(* PLC project 1000-tech-water, Неизвестно 1000-tech-water 1 *)
(* stored: creationDateTime 2022-06-13T20:45:02, productRelease 0, contentDescription 2022-06-20 Локальные испытания: выполнены Комплексные испытания: выполнены, modificationDateTime 2022-06-20T21:02:03, version 0, language ru-RU *)

PROGRAM Main
  VAR_EXTERNAL
    LT_Low : BOOL;
  END_VAR
  VAR
    LT_Low_f : BOOL;  (* Отфильтрованное значение *)
  END_VAR
  VAR_EXTERNAL
    LT_Middle : BOOL;
  END_VAR
  VAR
    LT_Middle_f : BOOL;  (* Отфильтрованное значение *)
  END_VAR
  VAR_EXTERNAL
    LT_Hight : BOOL;
  END_VAR
  VAR
    LT_Hight_f : BOOL;  (* Отфильтрованное значение *)
  END_VAR
  VAR_EXTERNAL
    HS_Auto : BOOL;
  END_VAR
  VAR
    HS_Auto_f : BOOL;  (* Отфильтрованное значение *)
  END_VAR
  VAR_EXTERNAL
    P_Speed_50 : BOOL;
  END_VAR
  VAR
    P_Speed_50L : BOOL;
  END_VAR
  VAR_EXTERNAL
    P_Speed_100 : BOOL;
  END_VAR
  VAR
    P_Speed_100L : BOOL;
  END_VAR
  VAR_EXTERNAL
    P_Start : BOOL;
  END_VAR
  VAR
    P_StartL : BOOL;
  END_VAR
  VAR_EXTERNAL
    LT_error : BOOL;
  END_VAR
  VAR
    LT_errorL : BOOL;
  END_VAR
  VAR_EXTERNAL
    LT_set : BOOL;
    PLC_state : WORD;
  END_VAR
  VAR
    TON0 : TON;
  END_VAR
  VAR CONSTANT
    TM_5S : TIME := T#5s;  (* Время 5 сек *)
  END_VAR
  VAR
    TON1 : TON;
    TON2 : TON;
    TON3 : TON;
  END_VAR
  VAR  (* added by the conversion: wires and edge detectors of the diagram *)
    _OR68_OUT : BOOL;
    _OR58_OUT : BOOL;
  END_VAR

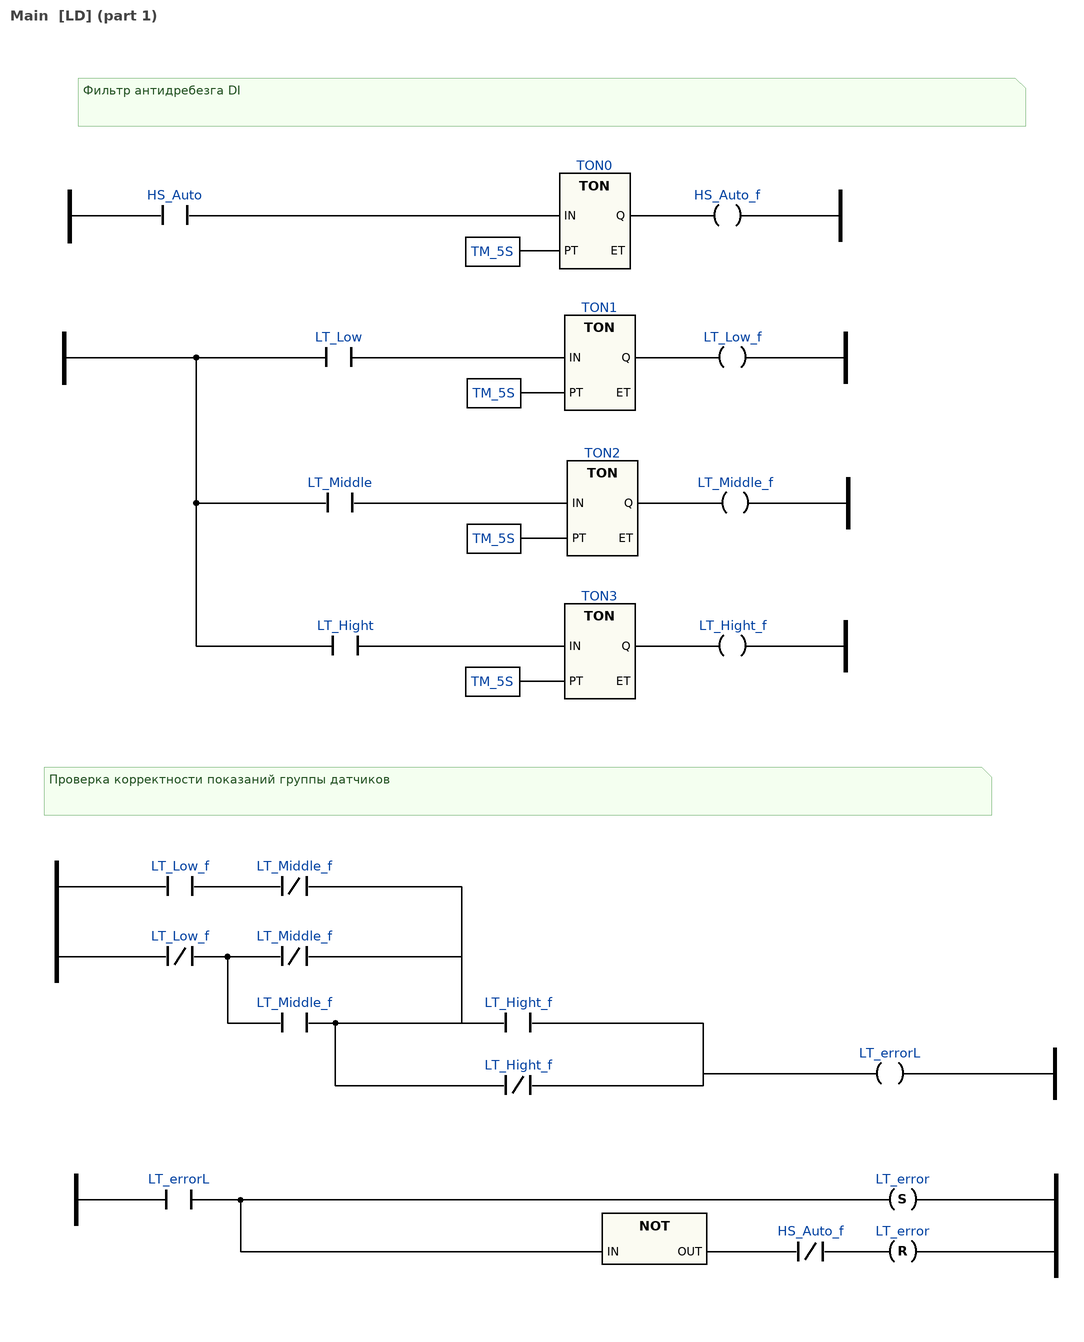
(* LD diagram, written out as Structured Text *)
(* Фильтр антидребезга DI *)
TON0(IN := HS_Auto, PT := TM_5S);
HS_Auto_f := TON0.Q;
TON1(IN := LT_Low, PT := TM_5S);
LT_Low_f := TON1.Q;
TON2(IN := LT_Middle, PT := TM_5S);
LT_Middle_f := TON2.Q;
TON3(IN := LT_Hight, PT := TM_5S);
LT_Hight_f := TON3.Q;
(* Проверка корректности показаний группы датчиков *)
LT_errorL := NOT LT_Low_f AND LT_Middle_f AND NOT LT_Hight_f OR (NOT LT_Low_f AND LT_Middle_f OR NOT LT_Low_f AND NOT LT_Middle_f OR LT_Low_f AND NOT LT_Middle_f) AND LT_Hight_f;
IF LT_errorL THEN LT_error := TRUE; END_IF;
IF NOT LT_errorL AND NOT HS_Auto_f THEN LT_error := FALSE; END_IF;
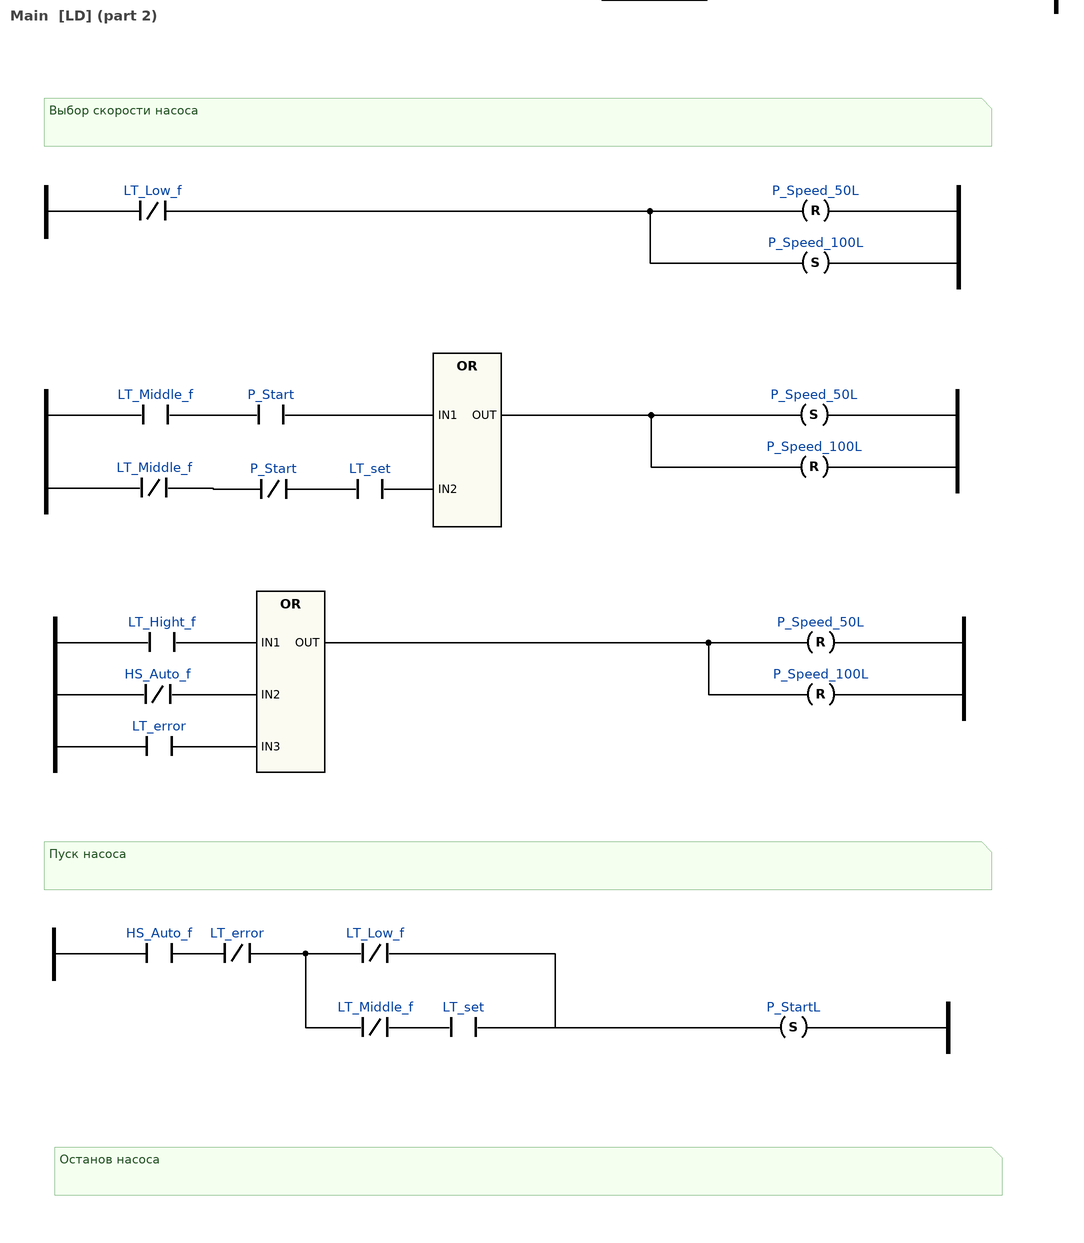
(* Выбор скорости насоса *)
IF NOT LT_Low_f THEN P_Speed_50L := FALSE; END_IF;
IF NOT LT_Low_f THEN P_Speed_100L := TRUE; END_IF;
_OR68_OUT := LT_Middle_f AND P_Start OR NOT LT_Middle_f AND NOT P_Start AND LT_set;
IF _OR68_OUT THEN P_Speed_50L := TRUE; END_IF;
IF _OR68_OUT THEN P_Speed_100L := FALSE; END_IF;
_OR58_OUT := LT_Hight_f OR NOT HS_Auto_f OR LT_error;
IF _OR58_OUT THEN P_Speed_50L := FALSE; END_IF;
IF _OR58_OUT THEN P_Speed_100L := FALSE; END_IF;
(* Пуск насоса *)
IF HS_Auto_f AND NOT LT_error AND (NOT LT_Low_f OR NOT LT_Middle_f AND LT_set) THEN P_StartL := TRUE; END_IF;
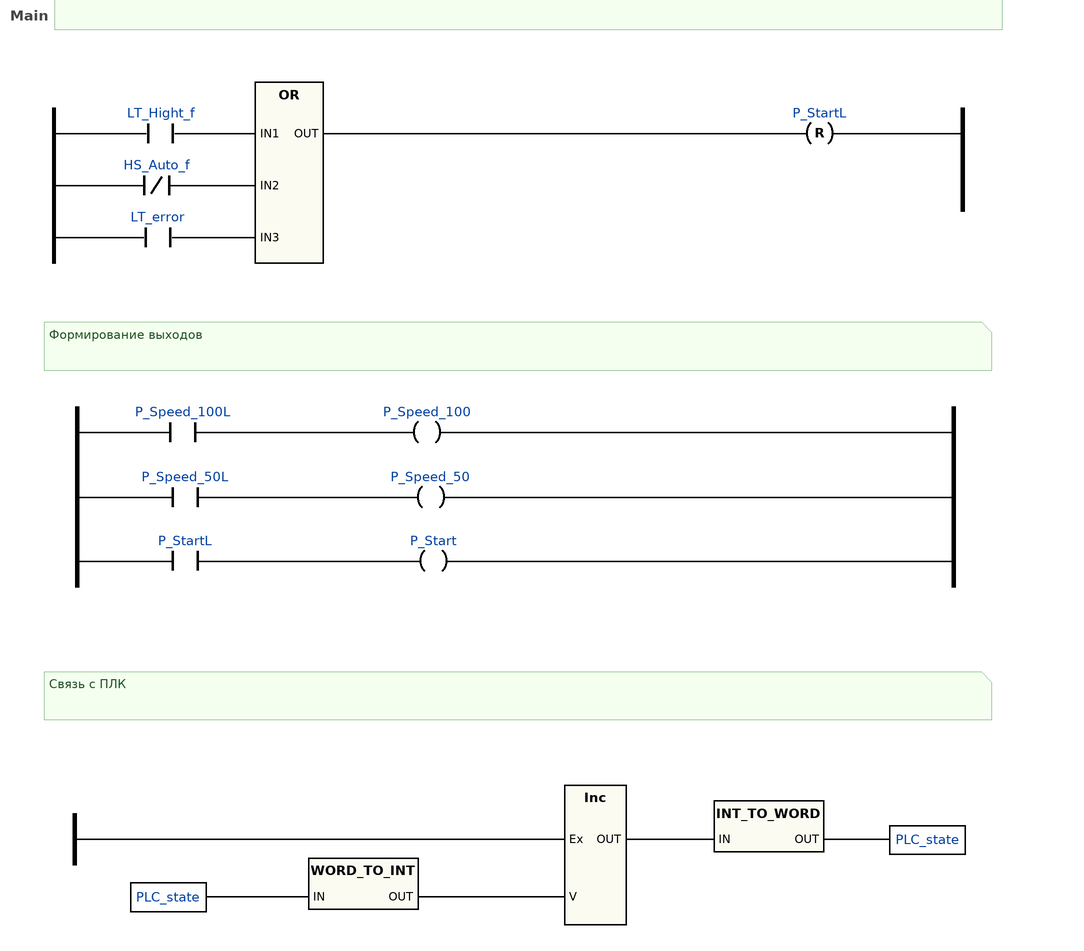
(* Останов насоса *)
IF LT_Hight_f OR NOT HS_Auto_f OR LT_error THEN P_StartL := FALSE; END_IF;
(* Формирование выходов *)
P_Speed_100 := P_Speed_100L;
P_Speed_50 := P_Speed_50L;
P_Start := P_StartL;
(* Связь с ПЛК *)
PLC_state := INT_TO_WORD(Inc(TRUE, WORD_TO_INT(PLC_state)));
END_PROGRAM

CONFIGURATION config
  VAR_GLOBAL
    LT_Low AT %IX1.0.1.1 : BOOL := FALSE;  (* Датчик нижнего уровня (1-LT-001) *)
    LT_Middle AT %IX1.1.1.1 : BOOL := FALSE;  (* Датчик среднего уровня (1-LT-002) *)
    LT_Hight AT %IX1.2.1.1 : BOOL := FALSE;  (* Датчик верхнего уровня (1-LT-003) *)
    HS_Auto AT %IX1.3.1.1 : BOOL := FALSE;  (* Переключатель Работа/Останов (1-HS-001) *)
    P_Speed_50 AT %QX5.0.1.1 : BOOL := FALSE;  (* Скорость 50% (Частотник для 1-P-001) *)
    P_Speed_100 AT %QX5.1.1.1 : BOOL := FALSE;  (* Скорость 100% (Частотник для 1-P-001) *)
    P_Start AT %QX5.2.1.1 : BOOL := FALSE;  (* Пуск/Стоп (Частотник для 1-P-001) *)
    LT_error AT %MX8.1.0 : BOOL := FALSE;  (* Ошибка датчиков уровней (признак) *)
    LT_set AT %MX8.1.1 : BOOL := FALSE;  (* Допустимый уровень опустошения бака (настройка) *)
    PLC_state AT %MW8.2.0 : WORD := 0;  (* Признак работы ПЛК *)
  END_VAR
  RESOURCE resource1 ON PLC
    TASK task0(INTERVAL := T#350ms, PRIORITY := 0);
    PROGRAM instance0 WITH task0 : Main;
  END_RESOURCE
END_CONFIGURATION
